// Mitsubishi GX Works2 project: 타이머 기본   PLC: Q03UDV

PROGRAM MAIN
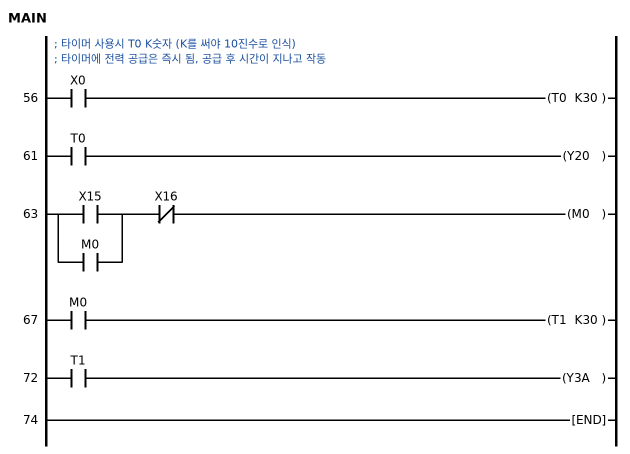
; 타이머 사용시 T0 K숫자 (K를 써야 10진수로 인식)
; 타이머에 전력 공급은 즉시 됨, 공급 후 시간이 지나고 작동
56    LD      X0
      OUT     T0 K30
61    LD      T0
      OUT     Y20
63    LD      X15
      OR      M0
      ANI     X16
      OUT     M0
67    LD      M0
      OUT     T1 K30
72    LD      T1
      OUT     Y3A
74    END
END_PROGRAM
